FUNCTION_BLOCK OthersDischargeValves (* Composite Function Block Type *)
  (* Standard: 61499-2 *)
  (* Version 0.0, 6/19/2026, Schneider Electric, template *)
  PACKAGE SE.Nereda;
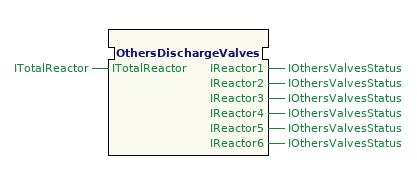
  SOCKETS
    ITotalReactor : ITotalReactor;
  END_SOCKETS
  PLUGS
    IReactor1 : IOthersValvesStatus;
    IReactor2 : IOthersValvesStatus;
    IReactor3 : IOthersValvesStatus;
    IReactor4 : IOthersValvesStatus;
    IReactor5 : IOthersValvesStatus;
    IReactor6 : IOthersValvesStatus;
  END_PLUGS
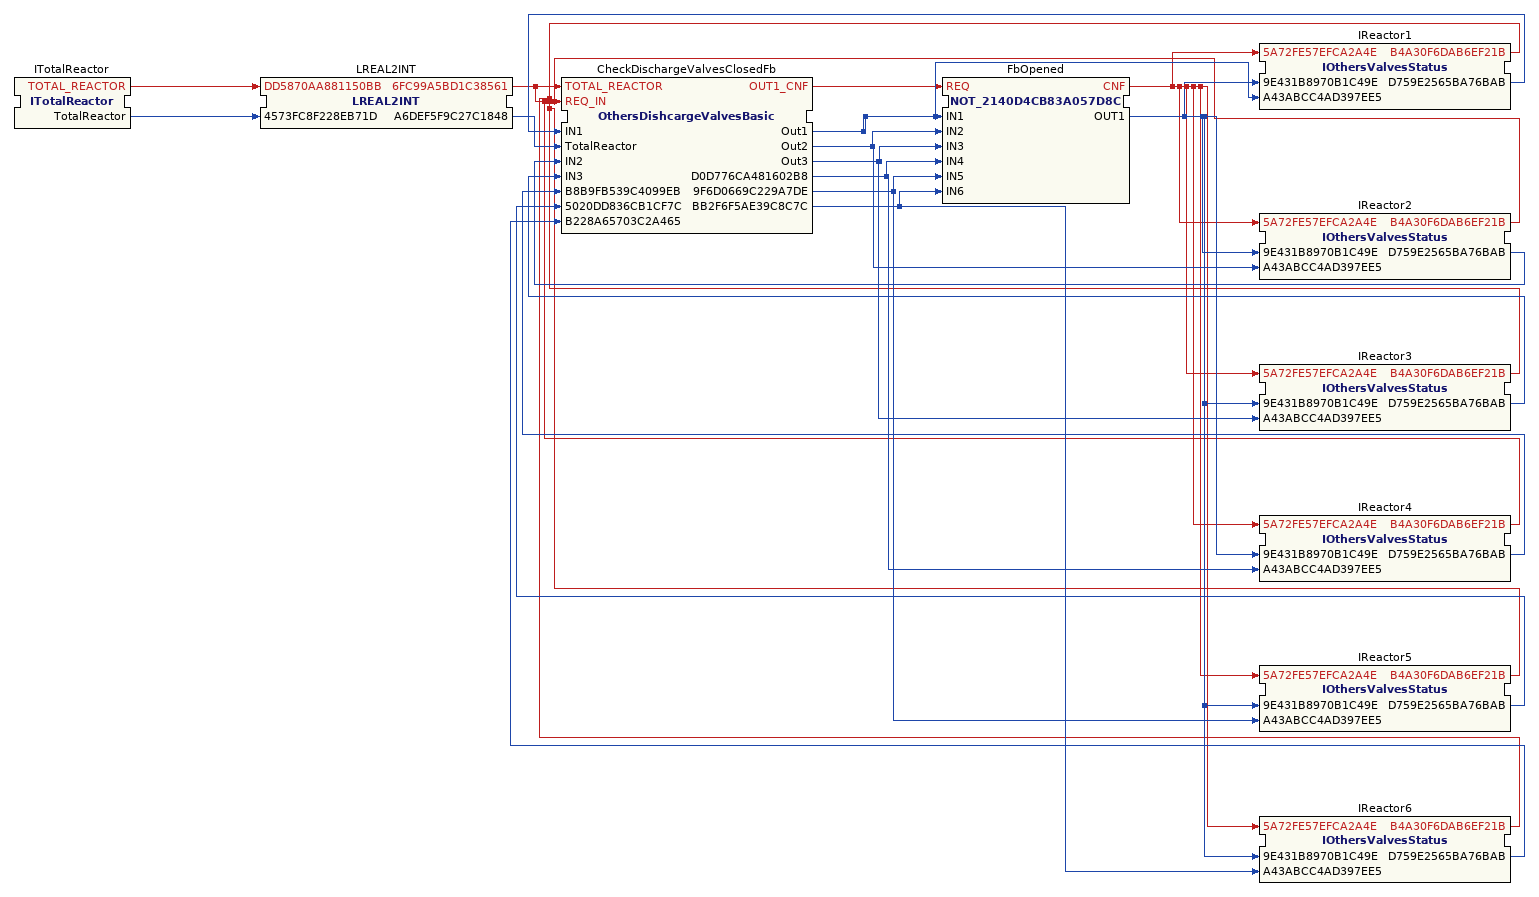
  (* 01 - FUNCTIONNAL INPUT INTERFACE *)
  (* 00 - INITIALIZATION *)
  (* 05 - LOGIC *)
  (* 03 - FIELD INTERFACE *)
  (* 02 - FUNCTIONNAL OUTPUT INTERFACE *)
  (* Others Valves Status *)
  (* 04 - CHILDREN *)
  (* 4A - TYPICALS *)
  FBS
    CheckDischargeValvesClosedFb : OthersDishcargeValvesBasic;
    FbOpened : NOT_2140D4CB83A057D8C; {SET_ATTRIBUTE(Configuration.GenericFBType.InterfaceParams, Runtime.Standard#CNT:=6;OUT${CNT$}:BOOL,BOOL,BOOL,BOOL,BOOL,BOOL)}
    LREAL2INT : LREAL2INT;
  END_FBS
  EVENT_CONNECTIONS
    LREAL2INT.6FC99A5BD1C38561 TO CheckDischargeValvesClosedFb.TOTAL_REACTOR;
    LREAL2INT.6FC99A5BD1C38561 TO CheckDischargeValvesClosedFb.REQ_IN;
    ITotalReactor.TOTAL_REACTOR TO LREAL2INT.DD5870AA881150BB;
    CheckDischargeValvesClosedFb.OUT1_CNF TO FbOpened.REQ;
    FbOpened.CNF TO IReactor1.5A72FE57EFCA2A4E;
    FbOpened.CNF TO IReactor2.5A72FE57EFCA2A4E;
    FbOpened.CNF TO IReactor3.5A72FE57EFCA2A4E;
    FbOpened.CNF TO IReactor4.5A72FE57EFCA2A4E;
    FbOpened.CNF TO IReactor5.5A72FE57EFCA2A4E;
    FbOpened.CNF TO IReactor6.5A72FE57EFCA2A4E;
    IReactor1.B4A30F6DAB6EF21B TO CheckDischargeValvesClosedFb.REQ_IN;
    IReactor2.B4A30F6DAB6EF21B TO CheckDischargeValvesClosedFb.REQ_IN;
    IReactor3.B4A30F6DAB6EF21B TO CheckDischargeValvesClosedFb.REQ_IN;
    IReactor4.B4A30F6DAB6EF21B TO CheckDischargeValvesClosedFb.REQ_IN;
    IReactor5.B4A30F6DAB6EF21B TO CheckDischargeValvesClosedFb.REQ_IN;
    IReactor6.B4A30F6DAB6EF21B TO CheckDischargeValvesClosedFb.REQ_IN;
  END_CONNECTIONS
  DATA_CONNECTIONS
    ITotalReactor.TotalReactor TO LREAL2INT.4573FC8F228EB71D;
    CheckDischargeValvesClosedFb.Out1 TO FbOpened.IN1;
    CheckDischargeValvesClosedFb.Out2 TO FbOpened.IN2;
    CheckDischargeValvesClosedFb.Out3 TO FbOpened.IN3;
    CheckDischargeValvesClosedFb.D0D776CA481602B8 TO FbOpened.IN4;
    CheckDischargeValvesClosedFb.9F6D0669C229A7DE TO FbOpened.IN5;
    CheckDischargeValvesClosedFb.BB2F6F5AE39C8C7C TO FbOpened.IN6;
    FbOpened.OUT1 TO IReactor1.9E431B8970B1C49E;
    FbOpened.OUT1 TO IReactor2.9E431B8970B1C49E;
    FbOpened.OUT1 TO IReactor3.9E431B8970B1C49E;
    FbOpened.OUT1 TO IReactor4.9E431B8970B1C49E;
    FbOpened.OUT1 TO IReactor5.9E431B8970B1C49E;
    FbOpened.OUT1 TO IReactor6.9E431B8970B1C49E;
    CheckDischargeValvesClosedFb.Out1 TO IReactor1.A43ABCC4AD397EE5;
    CheckDischargeValvesClosedFb.Out2 TO IReactor2.A43ABCC4AD397EE5;
    CheckDischargeValvesClosedFb.Out3 TO IReactor3.A43ABCC4AD397EE5;
    CheckDischargeValvesClosedFb.D0D776CA481602B8 TO IReactor4.A43ABCC4AD397EE5;
    CheckDischargeValvesClosedFb.9F6D0669C229A7DE TO IReactor5.A43ABCC4AD397EE5;
    CheckDischargeValvesClosedFb.BB2F6F5AE39C8C7C TO IReactor6.A43ABCC4AD397EE5;
    IReactor1.D759E2565BA76BAB TO CheckDischargeValvesClosedFb.IN1;
    LREAL2INT.A6DEF5F9C27C1848 TO CheckDischargeValvesClosedFb.TotalReactor;
    IReactor2.D759E2565BA76BAB TO CheckDischargeValvesClosedFb.IN2;
    IReactor3.D759E2565BA76BAB TO CheckDischargeValvesClosedFb.IN3;
    IReactor4.D759E2565BA76BAB TO CheckDischargeValvesClosedFb.B8B9FB539C4099EB;
    IReactor5.D759E2565BA76BAB TO CheckDischargeValvesClosedFb.5020DD836CB1CF7C;
    IReactor6.D759E2565BA76BAB TO CheckDischargeValvesClosedFb.B228A65703C2A465;
  END_CONNECTIONS
END_FUNCTION_BLOCK
